TYPE "udt_PAC3220"
VERSION : 0.1
// Block: udt_PAC3220
   STRUCT
      Voltage_L1 : Real;
      Voltage_L2 : Real;
      Voltage_L3 : Real;
      Current_L1 : Real;
      Current_L2 : Real;
      Current_L3 : Real;
      "AverageVoltageUL-L" : Real;
      AverageCurrent : Real;
      TotalActivePower : Real;
      TotalReactivePower : Real;
      TotalActiveEnergy : LReal;
      TotalApparentEnergy : LReal;
   END_STRUCT;

END_TYPE
